PROGRAM TEST
VAR
  _initDone : BOOL:= FALSE;
  _preparationsDone : BOOL:= FALSE;  
  _unitTestsDone : BOOL:= FALSE;
  
  
  //preparations
  
  //list tests here
  _bitFunctions_Test : FB_BitFunctions_Test;
  //...
  
END_VAR

IF _initDone = FALSE THEN
  Init();
  RETURN;
END_IF

IF _preparationsDone = FALSE THEN
  preparations();
  RETURN;
END_IF

//test
TcUnit.RUN();

_unitTestsDone := TcUnit.GVL_TcUnit.TcUnitRunner.AllTestSuitesFinished;

METHOD PUBLIC Init : BOOL
VAR_INPUT
END_VAR
VAR
    initResult              : BOOL;
END_VAR
Init:= FALSE;

// init to be done
initResult := TRUE;

// result
IF initResult THEN
  Init:= TRUE;
  _initDone:= TRUE;
END_IF
END_METHOD

METHOD PRIVATE preparations
VAR_STAT
END_VAR
VAR
  delayTON : TON := (IN:= FALSE);
END_VAR
_preparationsDone := TRUE;
END_METHOD

{attribute 'monitoring' := 'call'}
PROPERTY PUBLIC UnitTestsDone : BOOL
GET
UnitTestsDone:= _unitTestsDone;
END_GET
END_PROPERTY

END_PROGRAM

(* stored: Version 1.1.0.1, ProductVersion 3.1.4024.10
   POU TEST: Id {3687160c-057b-47bd-85ba-279fe0b8566e}, SpecialFunc None
   Folder _private: Id {e749bcbf-fa4f-4454-af58-9e964b4ad41c}
   Method Init: Id {0203137e-f26f-4371-9f12-ba46eb2b7bc0}
   Method preparations: Id {d8e006a1-25e7-41af-bed5-884bc17e7c08}
   Property UnitTestsDone: Id {13ea6760-ca09-4025-a657-7c70ff523b0c}
   Get Get: Id {c8549513-1e35-4300-bb13-f5749cb7acb7} *)
